# EPICS substitutions: lensApp/Db/beam.substitutions
file beam.tpl-db
{
    {
        LOCATION       = $(LOCATION)
        NLENS          = $(NLENS)
        ENERGY         = $(ENERGY)
    }
}
